(* CODESYS project canbus.remote.controller.20200324.01.project
   Description: Receives some incoming messages and echoes them with CAN-ID +1
   Company: 3S - Smart Software Solutions GmbH
   Version: 1.0.0.0
   Title: CAN Bus API Example
   Author: 3S - Smart Software Solutions GmbH

Project tree, tasks and I/O mapping:
  Device : Changsha-Cyber-MI-linux, Changsha Cyber-MI Co., Ltd., version 3.5.10.40
    application Application
      libraries: CAN API, 1.0.0.3 (3S - Smart Software Solutions GmbH); Standard, * (System); CAA CiA 405, * (CAA Technical Workgroup)
      task MainTask (cyclic, interval t#20ms, priority 1) calls prg_remote_controller
      global variables GVL
      CFC Example/
        program prg_remote_controller [CFC]
      ST Example/
        function block MsgProcessor_181_281 [ST]: ProcessMessage
    SoftMotion General Axis Pool
    CANbus_1 : CANbus, 3S - Smart Software Solutions GmbH, version 3.5.12.0
      CANopen_Manager : CANopen_Manager, 3S - Smart Software Solutions GmbH, version 3.5.10.0
          settings: ConfigVersion = 50659584
        Singleturn_Encoder_M36X8 : Singleturn Encoder M36X8, Kuebler GmbH, order no. 8.M36X8.XXCX.211X, version Revision=16#00000006, FileVersion=1.5
            settings: NODEIDSAVED = 1; SDO Timeout = 1000000; EXPERTSETTINGS = FALSE; Heartbeat-Producer Time = 200; PDO 16#1800.COBID = 16#00000181; Process by CANopenManager = TRUE; PDO 16#1801.COBID = 16#00000281; PDO 16#1801.Transmission Type = 16#01; Process by CANopenManager = TRUE; PDO 16#1802.COBID = 16#00000381; Process by CANopenManager = TRUE; Position Value.Subindex = 16#00; Speed Value 1.Subindex = 16#01; Position Value.Subindex = 16#00; SDO List.Set Guardtime.Index = 16#100C; SDO List.Set Guardtime.Subindex = 16#00; SDO List.Set Guardtime.Value = 16#00000000; SDO List.Set Guardtime.Size = 16; SDO List.Set Guardtime.AbortIfError = FALSE; SDO List.Set Guardtime.JumpToLine = FALSE; SDO List.Set Guardtime.Line = 0; SDO List.Set Lifetime.Index = 16#100D; SDO List.Set Lifetime.Subindex = 16#00; SDO List.Set Lifetime.Value = 16#00000000; SDO List.Set Lifetime.Size = 8; SDO List.Set Lifetime.AbortIfError = FALSE; SDO List.Set Lifetime.JumpToLine = FALSE; SDO List.Set Lifetime.Line = 0; SDO List.Set Heartbeat Producer.Index = 16#1017; SDO List.Set Heartbeat Producer.Subindex = 16#00; SDO List.Set Heartbeat Producer.Value = 16#000000C8; SDO List.Set Heartbeat Producer.Size = 16; SDO List.Set Heartbeat Producer.AbortIfError = FALSE; SDO List.Set Heartbeat Producer.JumpToLine = FALSE; SDO List.Set Heartbeat Producer.Line = 0; SDO List.Disable PDO.Index = 16#1800; SDO List.Disable PDO.Subindex = 16#01; SDO List.Disable PDO.Value = 16#80000181; SDO List.Disable PDO.Size = 32; SDO List.Disable PDO.AbortIfError = FALSE;
              SDO List.Disable PDO.JumpToLine = FALSE; SDO List.Disable PDO.Line = 0; SDO List.Set transmission type.Index = 16#1800; SDO List.Set transmission type.Subindex = 16#02; SDO List.Set transmission type.Value = 16#FF; SDO List.Set transmission type.Size = 8; SDO List.Set transmission type.AbortIfError = FALSE; SDO List.Set transmission type.JumpToLine = FALSE; SDO List.Set transmission type.Line = 0; SDO List.Set inhibit time.Index = 16#1800; SDO List.Set inhibit time.Subindex = 16#03; SDO List.Set inhibit time.Value = 16#0000; SDO List.Set inhibit time.Size = 16; SDO List.Set inhibit time.AbortIfError = FALSE; SDO List.Set inhibit time.JumpToLine = FALSE; SDO List.Set inhibit time.Line = 0; SDO List.Set event time.Index = 16#1800; SDO List.Set event time.Subindex = 16#05; SDO List.Set event time.Value = 16#0000; SDO List.Set event time.Size = 16; SDO List.Set event time.AbortIfError = FALSE; SDO List.Set event time.JumpToLine = FALSE; SDO List.Set event time.Line = 0; SDO List.Clear pdo mapping.Index = 16#1A00; SDO List.Clear pdo mapping.Subindex = 16#00; SDO List.Clear pdo mapping.Value = 16#0; SDO List.Clear pdo mapping.Size = 8; SDO List.Clear pdo mapping.AbortIfError = FALSE; SDO List.Clear pdo mapping.JumpToLine = FALSE; SDO List.Clear pdo mapping.Line = 0; SDO List.Set Mapping.Index = 16#1A00; SDO List.Set Mapping.Subindex = 16#01; SDO List.Set Mapping.Value = 16#60040020; SDO List.Set Mapping.Size = 32; SDO List.Set Mapping.AbortIfError = FALSE; SDO List.Set Mapping.JumpToLine = FALSE; SDO List.Set Mapping.Line = 0; SDO List.Set number of mappings.Index = 16#1A00; SDO List.Set number of mappings.Subindex = 16#00; SDO List.Set number of mappings.Value = 16#01;
              SDO List.Set number of mappings.Size = 8; SDO List.Set number of mappings.AbortIfError = FALSE; SDO List.Set number of mappings.JumpToLine = FALSE; SDO List.Set number of mappings.Line = 0; SDO List.Set and enable COB-ID.Index = 16#1800; SDO List.Set and enable COB-ID.Subindex = 16#01; SDO List.Set and enable COB-ID.Value = 16#00000181; SDO List.Set and enable COB-ID.Size = 32; SDO List.Set and enable COB-ID.AbortIfError = FALSE; SDO List.Set and enable COB-ID.JumpToLine = FALSE; SDO List.Set and enable COB-ID.Line = 0; SDO List.Disable PDO.Index = 16#1801; SDO List.Disable PDO.Subindex = 16#01; SDO List.Disable PDO.Value = 16#80000281; SDO List.Disable PDO.Size = 32; SDO List.Disable PDO.AbortIfError = FALSE; SDO List.Disable PDO.JumpToLine = FALSE; SDO List.Disable PDO.Line = 0; SDO List.Set transmission type.Index = 16#1801; SDO List.Set transmission type.Subindex = 16#02; SDO List.Set transmission type.Value = 16#01; SDO List.Set transmission type.Size = 8; SDO List.Set transmission type.AbortIfError = FALSE; SDO List.Set transmission type.JumpToLine = FALSE; SDO List.Set transmission type.Line = 0; SDO List.Set inhibit time.Index = 16#1801; SDO List.Set inhibit time.Subindex = 16#03; SDO List.Set inhibit time.Value = 16#0000; SDO List.Set inhibit time.Size = 16; SDO List.Set inhibit time.AbortIfError = FALSE; SDO List.Set inhibit time.JumpToLine = FALSE; SDO List.Set inhibit time.Line = 0; SDO List.Set event time.Index = 16#1801; SDO List.Set event time.Subindex = 16#05; SDO List.Set event time.Value = 16#0000; SDO List.Set event time.Size = 16; SDO List.Set event time.AbortIfError = FALSE; SDO List.Set event time.JumpToLine = FALSE; SDO List.Set event time.Line = 0; SDO List.Clear pdo mapping.Index = 16#1A01;
              SDO List.Clear pdo mapping.Subindex = 16#00; SDO List.Clear pdo mapping.Value = 16#0; SDO List.Clear pdo mapping.Size = 8; SDO List.Clear pdo mapping.AbortIfError = FALSE; SDO List.Clear pdo mapping.JumpToLine = FALSE; SDO List.Clear pdo mapping.Line = 0; SDO List.Set Mapping.Index = 16#1A01; SDO List.Set Mapping.Subindex = 16#01; SDO List.Set Mapping.Value = 16#60300110; SDO List.Set Mapping.Size = 32; SDO List.Set Mapping.AbortIfError = FALSE; SDO List.Set Mapping.JumpToLine = FALSE; SDO List.Set Mapping.Line = 0; SDO List.Set number of mappings.Index = 16#1A01; SDO List.Set number of mappings.Subindex = 16#00; SDO List.Set number of mappings.Value = 16#01; SDO List.Set number of mappings.Size = 8; SDO List.Set number of mappings.AbortIfError = FALSE; SDO List.Set number of mappings.JumpToLine = FALSE; SDO List.Set number of mappings.Line = 0; SDO List.Set and enable COB-ID.Index = 16#1801; SDO List.Set and enable COB-ID.Subindex = 16#01; SDO List.Set and enable COB-ID.Value = 16#00000281; SDO List.Set and enable COB-ID.Size = 32; SDO List.Set and enable COB-ID.AbortIfError = FALSE; SDO List.Set and enable COB-ID.JumpToLine = FALSE; SDO List.Set and enable COB-ID.Line = 0; SDO List.Disable PDO.Index = 16#1802; SDO List.Disable PDO.Subindex = 16#01; SDO List.Disable PDO.Value = 16#80000381; SDO List.Disable PDO.Size = 32; SDO List.Disable PDO.AbortIfError = FALSE; SDO List.Disable PDO.JumpToLine = FALSE; SDO List.Disable PDO.Line = 0; SDO List.Set transmission type.Index = 16#1802; SDO List.Set transmission type.Subindex = 16#02; SDO List.Set transmission type.Value = 16#FF; SDO List.Set transmission type.Size = 8; SDO List.Set transmission type.AbortIfError = FALSE; SDO List.Set transmission type.JumpToLine = FALSE;
              SDO List.Set transmission type.Line = 0; SDO List.Set inhibit time.Index = 16#1802; SDO List.Set inhibit time.Subindex = 16#03; SDO List.Set inhibit time.Value = 16#0000; SDO List.Set inhibit time.Size = 16; SDO List.Set inhibit time.AbortIfError = FALSE; SDO List.Set inhibit time.JumpToLine = FALSE; SDO List.Set inhibit time.Line = 0; SDO List.Set event time.Index = 16#1802; SDO List.Set event time.Subindex = 16#05; SDO List.Set event time.Value = 16#0000; SDO List.Set event time.Size = 16; SDO List.Set event time.AbortIfError = FALSE; SDO List.Set event time.JumpToLine = FALSE; SDO List.Set event time.Line = 0; SDO List.Clear pdo mapping.Index = 16#1A02; SDO List.Clear pdo mapping.Subindex = 16#00; SDO List.Clear pdo mapping.Value = 16#0; SDO List.Clear pdo mapping.Size = 8; SDO List.Clear pdo mapping.AbortIfError = FALSE; SDO List.Clear pdo mapping.JumpToLine = FALSE; SDO List.Clear pdo mapping.Line = 0; SDO List.Set Mapping.Index = 16#1A02; SDO List.Set Mapping.Subindex = 16#01; SDO List.Set Mapping.Value = 16#60040020; SDO List.Set Mapping.Size = 32; SDO List.Set Mapping.AbortIfError = FALSE; SDO List.Set Mapping.JumpToLine = FALSE; SDO List.Set Mapping.Line = 0; SDO List.Set number of mappings.Index = 16#1A02; SDO List.Set number of mappings.Subindex = 16#00; SDO List.Set number of mappings.Value = 16#01; SDO List.Set number of mappings.Size = 8; SDO List.Set number of mappings.AbortIfError = FALSE; SDO List.Set number of mappings.JumpToLine = FALSE; SDO List.Set number of mappings.Line = 0; SDO List.Set and enable COB-ID.Index = 16#1802; SDO List.Set and enable COB-ID.Subindex = 16#01; SDO List.Set and enable COB-ID.Value = 16#00000381; SDO List.Set and enable COB-ID.Size = 32;
              SDO List.Set and enable COB-ID.AbortIfError = FALSE; SDO List.Set and enable COB-ID.JumpToLine = FALSE; SDO List.Set and enable COB-ID.Line = 0; ConfigVersion = 50659584
            unmapped channels: Position Value, Speed Value 1, Position Value
*)

// Device/Application/GVL
VAR_GLOBAL
//181帧变量
	xStart:BOOL := FALSE;  //启动
	xHorn:BOOL := FALSE;  //喇叭
	xEngStart:BOOL := FALSE; //发动机启动
//其它变量定义

//281帧变量
	bSpeed:BYTE := 0; //速度
	bRot: BYTE := 0;  //转向
//其它变量定义
	
END_VAR

// Device/Application/CFC Example/prg_remote_controller
/// Receives messages with CobIds ranging from 16#500 to 16#550 and echoes them back with CobId +1
PROGRAM prg_remote_controller
VAR
	driver29bit 	: CAN.CANDriver_29bit;
	                                
	areaReceiver	: CAN.CANAreaReceiver;
	singleReceiver	: CAN.CANSingleIdReceiver;
	diagnosis		: CAN.CANBusDiagnosis;
	
	msgProcessor	: MsgProcessor_181_281;
END_VAR
VAR // added by the converter: edge detectors and wires of the graphical bodies
    _s1 : CAN.DRIVER_CONFIG;
    _s2 : CAN.RECEIVER_AREA;
    _s3 : CAN.DIAGNOSIS_INFO;
    _s4 : CAN.RECEIVER_SINGLE_ID;
END_VAR

// compose _s1 : CAN.DRIVER_CONFIG
_s1.usiNetwork := 0;
_s1.uiBaudrate := 250;
_s1.ctMessages := 100;
driver29bit(xEnable := TRUE, DriverConfig := _s1); // CAN.CANDriver_29bit
// compose _s2 : CAN.RECEIVER_AREA
_s2.dwIdStart := 16#181;
_s2.dwIdEnd := 16#281;
_s2.xRTRValue := false;
_s2.xRTRMask := false;
_s2.xTransmitValue := false;
_s2.xTransmitMask := true;
areaReceiver(itfCANDriver := driver29bit, Area := _s2, itfMsgProcessor := msgProcessor, tTimeLimit := t#5ms); // CAN.CANAreaReceiver
singleReceiver(SingleId := _s4); // CAN.CANSingleIdReceiver
diagnosis(itfCANDriver := driver29bit, DiagnosticInfo := _s3); // CAN.CANBusDiagnosis
// compose _s3 : CAN.DIAGNOSIS_INFO
msgProcessor(CANdriver := driver29bit); // MsgProcessor_181_281
// compose _s4 : CAN.RECEIVER_SINGLE_ID
_s4.dwCanId := 16#280;
_s4.xRTRValue := false;
_s4.xRTRMask := false;
_s4.x29BitIdValue := false;
_s4.x29BitIdMask := false;
_s4.xTransmitValue := false;
_s4.xTransmitMask := true;
_s4.xAlwaysNewest := true;

END_PROGRAM

// Device/Application/ST Example/MsgProcessor_181_281
/// MsgProcessor_Echo is the implimentation of IMessageProcessor. 
/// MsgProcessor_Echo simply counts all incoming messages and echos them with CobId +1
FUNCTION_BLOCK MsgProcessor_181_281 IMPLEMENTS CAN.IMessageProcessor
VAR_IN_OUT
	CANdriver	: CAN.CANDriver_29bit;
END_VAR
VAR_OUTPUT
END_VAR
VAR
	_pCANdriver : POINTER TO CAN.CANDriver_29bit;
END_VAR

_pCANdriver := ADR(CANdriver);

METHOD ProcessMessage
VAR_IN_OUT
	(* The messages received by the receiver *)
	Message	: CAN.RxMessage;
END_VAR
VAR
	id:UDINT;
	data:BYTE;
END_VAR
IF _pCANdriver = 0 THEN
	RETURN;
END_IF

id := Message.udiCanID;

IF id = 16#181 THEN
	data := Message.abyData[0];
	gvl.xStart := data.0;
	gvl.xHorn := data.1;
	//其它变量赋值
	
ELSIF id = 16#281 THEN
	gvl.bSpeed := Message.abyData[0];
	gvl.bRot := Message.abyData[1];
	//其它变量赋值
	
END_IF
END_METHOD

END_FUNCTION_BLOCK
